FUNCTION_BLOCK FILE_WRITER_7 (* Writes equation coeficients to a file (7 coef) *)
  (* Standard: 61499-2 *)
  (* Version 1.0, 23-03-12, GASR, Universidade do Estado de Santa Catarina *)
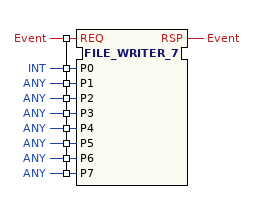
  EVENT_INPUT
    REQ WITH P0, P1, P2, P3, P4, P5, P6, P7; (* Request file storage *)
  END_EVENT
  EVENT_OUTPUT
    RSP; (* Finished operation *)
  END_EVENT
  VAR_INPUT
    P0 : INT; (* Process/equation id *)
    P1 : ANY; (* Coeficient 1 *)
    P2 : ANY; (* Coeficient 2 *)
    P3 : ANY; (* Coeficient 3 *)
    P4 : ANY; (* Coeficient 4 *)
    P5 : ANY; (* Coeficient 5 *)
    P6 : ANY; (* Coeficient 6 *)
    P7 : ANY; (* Coeficient 7 *)
  END_VAR
  SERVICE FILE_WRITER_7/MACHINE (* Coeficient file storage service *)
    SEQUENCE normal_establishment
      FILE_WRITER_7.REQ(P0,P1,P2,P3,P4,P5,P6,P7) -> MACHINE.write-file();
      MACHINE.response() -> FILE_WRITER_7.RSP();
    END_SEQUENCE
  END_SERVICE
END_FUNCTION_BLOCK
